Yaskawa INFORM job: STKMISS.JBI

/JOB
//NAME STKMISS
///FOLDERNAME SpeedbotUnStack
//POS
///NPOS 0,0,0,0,0,0
//INST
///DATE 2025/04/20 20:38
///ATTR SC,RW
///GROUP1 RB1
///LVARS 10,10,10,10,10,10,0,0
NOP
'@Part Id
GETARG LD000 IARG#(1)
SET D070 LD000
SET B069 0
'SKILLSND "UnStackMiss"
END
